// TIA Portal V20 export
FUNCTION_BLOCK "Oil"   // FB8, LAD
{ S7_Optimized_Access := 'TRUE' }
// stored: MemoryReserve 100, SetENOAutomatically false
   VAR_INPUT
      Safety_OK : Bool;
      Pump_status : Bool;
      Pump_error : Bool;
      Pallette_Moving : Bool;
   END_VAR
   VAR_OUTPUT
      Pump : Bool;
      Main_Valve : Bool;
      Preparation_Valve : Bool;
      Nozzle_Valve : Bool;
      Pump_Volume_Output : Int;
   END_VAR
   VAR
      Pump_Reset { S7_SetPoint := 'True'} : TON_TIME;
      Pump_Volume { S7_SetPoint := 'True'} : Real;
      Oil_Station_Enable : Bool;
   END_VAR
   VAR_TEMP
      tmp : Int;
   END_VAR
BEGIN

REGION Network 1
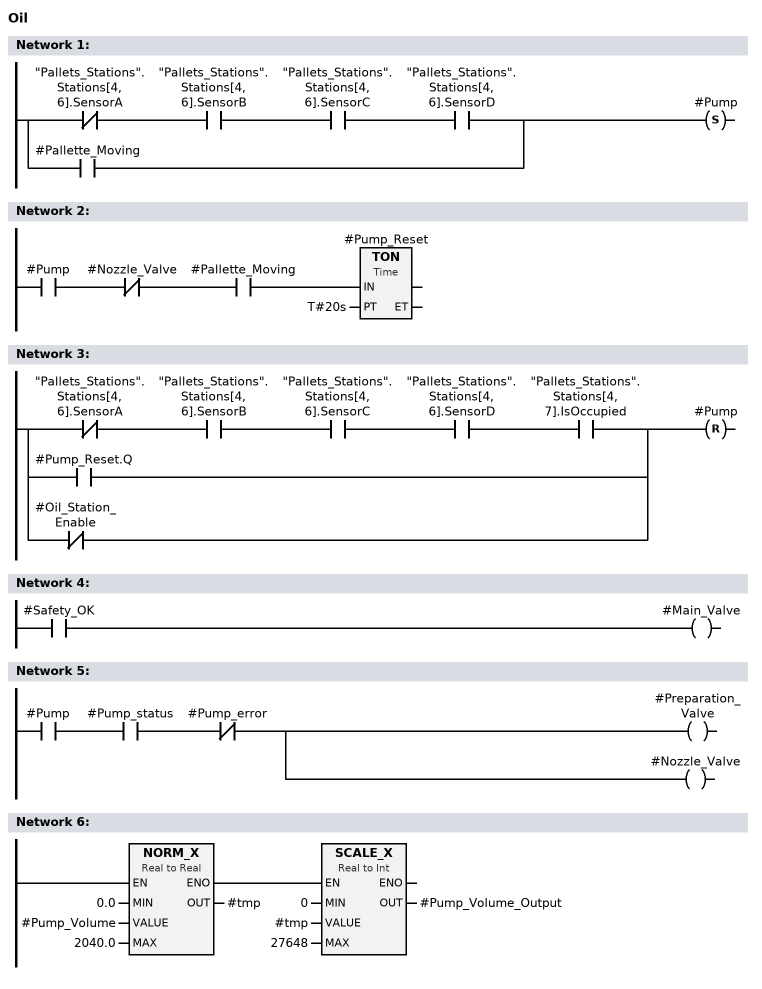
   RUNG wire#powerrail
      I_Contact( "Pallets_Stations".Stations[4, 6].SensorA )
      Contact( "Pallets_Stations".Stations[4, 6].SensorB )
      Contact( "Pallets_Stations".Stations[4, 6].SensorC )
      Contact( "Pallets_Stations".Stations[4, 6].SensorD )
      wire#w1
      S_Coil( #Pump )
   END_RUNG
   RUNG wire#powerrail
      Contact( #Pallette_Moving )
   END_RUNG wire#w1
   // the same network as SCL:
   IF (NOT "Pallets_Stations".Stations[4, 6].SensorA AND "Pallets_Stations".Stations[4, 6].SensorB AND "Pallets_Stations".Stations[4, 6].SensorC AND "Pallets_Stations".Stations[4, 6].SensorD) OR #Pallette_Moving THEN
       #Pump := TRUE;
   END_IF;
END_REGION

REGION Network 2
   RUNG wire#powerrail
      Contact( #Pump )
      I_Contact( #Nozzle_Valve )
      Contact( #Pallette_Moving )
      { S7_Templates := "time_type := Time" } #Pump_Reset.TON(pt := T#20s, et =>)
   END_RUNG
   // the same network as SCL:
   #Pump_Reset(IN := #Pump AND NOT #Nozzle_Valve AND #Pallette_Moving, PT := T#20s);   // TON
END_REGION

REGION Network 3
   RUNG wire#powerrail
      I_Contact( "Pallets_Stations".Stations[4, 6].SensorA )
      Contact( "Pallets_Stations".Stations[4, 6].SensorB )
      Contact( "Pallets_Stations".Stations[4, 6].SensorC )
      Contact( "Pallets_Stations".Stations[4, 6].SensorD )
      Contact( "Pallets_Stations".Stations[4, 7].IsOccupied )
      wire#w1
      R_Coil( #Pump )
   END_RUNG
   RUNG wire#powerrail
      Contact( #Pump_Reset.Q )
   END_RUNG wire#w1
   RUNG wire#powerrail
      I_Contact( #Oil_Station_Enable )
   END_RUNG wire#w1
   // the same network as SCL:
   IF (NOT "Pallets_Stations".Stations[4, 6].SensorA AND "Pallets_Stations".Stations[4, 6].SensorB AND "Pallets_Stations".Stations[4, 6].SensorC AND "Pallets_Stations".Stations[4, 6].SensorD AND "Pallets_Stations".Stations[4, 7].IsOccupied) OR #Pump_Reset.Q OR NOT #Oil_Station_Enable THEN
       #Pump := FALSE;
   END_IF;
END_REGION

REGION Network 4
   RUNG wire#powerrail
      Contact( #Safety_OK )
      Coil( #Main_Valve )
   END_RUNG
   // the same network as SCL:
   #Main_Valve := #Safety_OK;
END_REGION

REGION Network 5
   RUNG wire#powerrail
      Contact( #Pump )
      Contact( #Pump_status )
      I_Contact( #Pump_error )
      wire#w1
      Coil( #Preparation_Valve )
   END_RUNG
   RUNG wire#w1
      Coil( #Nozzle_Valve )
   END_RUNG
   // the same network as SCL:
   #Preparation_Valve := #Pump AND #Pump_status AND NOT #Pump_error;
   #Nozzle_Valve := #Preparation_Valve;
END_REGION

REGION Network 6
   RUNG wire#powerrail
      { S7_Templates := "[SrcType := Real, DestType := Real]" } Normalize(min := 0.0, value := #Pump_Volume, max := 2040.0, out => #tmp)
      { S7_Templates := "[SrcType := Real, DestType := Int]" } Scale(min := 0, value := #tmp, max := 27648, out => #Pump_Volume_Output)
   END_RUNG
   // the same network as SCL:
   #tmp := NORM_X(MIN := 0.0, VALUE := #Pump_Volume, MAX := 2040.0);
   #Pump_Volume_Output := SCALE_X(MIN := 0, VALUE := #tmp, MAX := 27648);
END_REGION
END_FUNCTION_BLOCK
